(* IEC 61131-3 sources: Kur_TemplateProject_v1/TestPanelV1.fbsproj/MyController.device.xml.v3^/Plc Logic.plclogic.xml.v3^/Application.application.xml.v3^/04_Programs, 1 file *)

(* ---- PRG_Main.prg.st ---- *)
PROGRAM PRG_Main
VAR
	// Deafult vars
	start     : Button;
	stop      : Button;
	reset     : EmergencyStop;
	emergency : EmergencyStop;

	// system vars (like motors, vars, ....)

END_VAR

// --------- CHECK StATUS -----
Machine.AxisOk		:= (DRV1.Axis.etAxisState <> 0);
Machine.BusOk		:= TRUE;
Machine.HomeOk		:= TRUE;
Machine.PowerOk		:= TRUE;
Machine.SafetyOk	:= TRUE;
